FUNCTION_BLOCK T_RoboConnect_WhenCalledWithLowTimeout_FailsConnection EXTENDS T_UnitTestBase
VAR
  robot : I_RoboConnect;
  timeOutTimer : TON;
  myTestState, prevState : (INIT, ARRANGE, ACT, ASSERT) := INIT;
  expected, actual : BOOL;
  counter : UINT;
END_VAR

CASE myTestState OF
  INIT:
    StateChanged();
    myTestState := ARRANGE;

  ARRANGE:
    StateChanged();

    expected := FALSE;
    myTestState := ACT;

  ACT:
    robot.Connect();
    myTestState := ASSERT;

  ASSERT:

    IF timeOutTimer.Q THEN
      actual := robot.Connected;
      assertion.AssertEquals_BOOL(expected, actual, 'IsConnected := FALSE');
      TestFinished();
      myTestState := INIT;
      robot.Disconnect();
    END_IF

END_CASE

timeOutTimer(IN := myTestState = ASSERT);

METHOD FB_init : BOOL
VAR_INPUT
  bInitRetains : BOOL; // if TRUE, the retain variables are initialized (warm start / cold start)
  bInCopyCode : BOOL; // if TRUE, the instance afterwards gets moved into the copy code (online change)
  TestSuite : tcl_SimpleUnitTestLibrary.I_TestSuite;
  robot : I_TcRobot;
  timeout : TIME;
END_VAR
THIS^.robot := robot;
THIS^.timeOutTimer.PT := timeout;
END_METHOD

METHOD PRIVATE StateChanged : BOOL
IF  myTestState = prevState THEN
  RETURN;
END_IF

prevState := myTestState;
StateChanged := TRUE;
END_METHOD

METHOD WaitForCycles : BOOL
VAR_INPUT
  maxCount : UINT;
END_VAR
counter := counter + 1;

IF counter = maxCount THEN
  counter := 0;
  WaitForCycles := TRUE;
END_IF
END_METHOD

END_FUNCTION_BLOCK

(* stored: Version 1.1.0.1
   POU T_RoboConnect_WhenCalledWithLowTimeout_FailsConnection: Id {807435e8-1c12-4909-8c7d-de689b94c80c}, SpecialFunc None
   Method FB_init: Id {5e070720-d7b0-485d-9126-850600772560}
   Method StateChanged: Id {71a88de3-7ae7-451c-b20f-40e743620782}
   Method WaitForCycles: Id {289ac53a-a335-437c-90a3-63ccd2de0a51} *)
